{attribute 'linkalways'} 
{attribute 'no_explicit_call' := 'This FB is a CLASS and must be accessed using methods or properties'}
{attribute 'enable_dynamic_creation'}
FUNCTION_BLOCK InputPortAddedEvent EXTENDS Disposable IMPLEMENTS I_InputPortAddedEvent
VAR
	_target : I_InputPort;
END_VAR

METHOD FB_init : BOOL
VAR_INPUT
	bInitRetains : BOOL; // if TRUE, the retain variables are initialized (warm start / cold start)
	bInCopyCode : BOOL;  // if TRUE, the instance afterwards gets moved into the copy code (online change)
	Target : I_InputPort;
END_VAR
THIS^._target := Target;
END_METHOD

PROPERTY PUBLIC Target : I_InputPort
GET
Target := _target;
END_GET
END_PROPERTY

END_FUNCTION_BLOCK

(* stored: Version 1.1.0.1, ProductVersion 3.1.4024.13
   POU InputPortAddedEvent: Id {f4a658e3-acc8-40b9-bf4a-bad2bc051631}, SpecialFunc None
   Folder Constructor: Id {6ade57b7-682e-4388-beca-08dbdcb648e2}
   Method FB_init: Id {4515e023-359d-493d-a337-c1c5fc49aac1}
   Property Target: Id {d7a7b31e-4b08-47c9-bf20-1d1e2f1402ca}
   Get Get: Id {87b6ca8c-9a24-4b19-9675-662c9a852499} *)
